{attribute 'no_explicit_call' := 'do not call this POU directly'} 
FUNCTION_BLOCK FB_LoggerProxy IMPLEMENTS I_Logger
VAR_INPUT
END_VAR
VAR_OUTPUT
END_VAR
VAR
	stHead    : ST_LoggerNode; // static head element
END_VAR

//FB_Exit muss explizit implementiert werden. Wenn es eine Implementierung gibt, dann wird 
//die Methode aufgerufen, bevor die Steuerung den Code der Funktionsbaustein-Instanz entfernt
//(impliziter Aufruf. Der Rückgabewert wird nicht ausgewertet.
METHOD FB_Exit: BOOL
VAR_INPUT    
bInCopyCode: BOOL;  // TRUE: Die Exit-Methode wird aufgerufen, um die Instanz zu verlassen, die hinterher kopiert wird Online-Change).  
END_VAR
M_Clear();
END_METHOD

METHOD M_Attach : BOOL
VAR_INPUT
    iLogger : I_Logger;
END_VAR
VAR
    pHead     : POINTER TO ST_LoggerNode := ADR(stHead);
    pCurrent  : POINTER TO ST_LoggerNode;
END_VAR
// invalid input
IF iLogger = 0 THEN
    RETURN(FALSE);
END_IF

// first node check
IF pHead^.iLogger = 0 THEN
    pHead^.iLogger := iLogger;
    pHead^.pNext := 0;
    RETURN(TRUE);
END_IF

// traverse list to check duplicates
pCurrent := pHead;
WHILE pCurrent^.pNext <> 0 DO
    IF pCurrent^.iLogger = iLogger THEN
        RETURN(FALSE); // already attached
    END_IF
    pCurrent := pCurrent^.pNext;
END_WHILE

// check last node
IF pCurrent^.iLogger = iLogger THEN
    RETURN(FALSE);
END_IF

// add new node
pCurrent^.pNext := __NEW(ST_LoggerNode);
IF pCurrent^.pNext = 0 THEN
    RETURN(FALSE);
END_IF
pCurrent^.pNext^.iLogger := iLogger;
pCurrent^.pNext^.pNext := 0;

RETURN(TRUE);
END_METHOD

METHOD PUBLIC M_Clear : BOOL
VAR_INPUT
END_VAR
VAR
    pCurrent : POINTER TO ST_LoggerNode;
    pNext    : POINTER TO ST_LoggerNode;
END_VAR
pCurrent := stHead.pNext; // start after head
WHILE pCurrent <> 0 DO
    pNext := pCurrent^.pNext; // store next pointer
    __DELETE(pCurrent);       // free current
    pCurrent := pNext;
END_WHILE

stHead.iLogger := 0;
stHead.pNext := 0;

M_Clear := TRUE;
END_METHOD

METHOD M_Log : BOOL
VAR_INPUT
	fbMessage	: FB_Message;
END_VAR
VAR
    pCurrent : POINTER TO ST_LoggerNode:= ADR(stHead);
END_VAR
WHILE pCurrent <> 0 DO
    pCurrent^.iLogger.M_Log(fbMessage);
    pCurrent := pCurrent^.pNext;
END_WHILE
M_Log := TRUE;
END_METHOD

END_FUNCTION_BLOCK

(* stored: Version 1.1.0.1
   POU FB_LoggerProxy: Id {c92161d9-49ae-4c50-bdac-f079e9b056c0}, SpecialFunc None
   Method FB_Exit: Id {5ffdbfed-bc35-4ea0-a3e2-08b0a045fdd8}
   Method M_Attach: Id {a672c9f6-c6e5-42cc-9e0b-921d3f608c6a}
   Method M_Clear: Id {e2bb2554-8db9-48a3-bb8b-1e817023fd88}
   Method M_Log: Id {eb21a125-c7d6-460d-84cb-3d1cb4ea2fdf} *)
